FUNCTION_BLOCK PickerContainer EXTENDS ZCore.ObjectContainer
VAR_INPUT
END_VAR
VAR_OUTPUT
END_VAR
VAR
  {attribute 'hide'}
  _parent : REFERENCE TO PickerUnit;
END_VAR

{attribute 'hide' }
METHOD FB_init : BOOL
VAR_INPUT
	bInitRetains : BOOL; // if TRUE, the retain variables are initialized (warm start / cold start)
	bInCopyCode : BOOL;  // if TRUE, the instance afterwards gets moved into the copy code (online change)
  unit : REFERENCE TO PickerUnit;
END_VAR
_parent REF= unit;
END_METHOD

END_FUNCTION_BLOCK

(* stored: Version 1.1.0.1
   POU PickerContainer: Id {41f82e27-e9a7-4f3c-81df-9f370712b1f6}, SpecialFunc None
   Method FB_init: Id {0122d4e3-eab8-4c93-90a8-c11043f50d41} *)
